PROGRAM OLD_MAIN
VAR
	fb_IndraDrive	: fbIndraDrive;
	stAmsNetId	AT %I*	: AMSNETID;
	nPort	AT %I* : WORD;
	stCommands: ST_AXIS_COMMAND;
	stStatus: ST_AXIS_STATUS;
	nMasterAxisPosition AT %I* : DINT;
	nAdditivePositionSetpoiunt AT %Q* : DINT;
	fMasterAxisPosition : LREAL;
	fAdditivePositionSetpoint : LREAL;
	fDiffPosition :LREAL;
	dLatchedPosition AT %I*:DINT;
	eTargetState: TARGET_STATE_MACHINE;
	bExecute: BOOL := FALSE;
	bEnable:BOOL:=FALSE;
	bEnabled:BOOL:=FALSE;
	bReset:BOOL:=FALSE;
    fbModePhase:FB_ModePhasing;	
	fAccelerationDefault:LREAL:=0.005;
	fSetVelToDriveRaw:LREAL;
	bBrakeFreewheelOn AT %Q*: BOOL;
	bBrakeLockedOn AT %Q*: BOOL;
    inputDummy AT %I*: BOOL;
	inputDigSens1 AT %I*: BOOL;
	inputDigSens2 AT %I*: BOOL;
	nMaxMotorTemperature: INT:= 50;
	fbBrakeTorque: FB_BrakeTorque;
	
END_VAR

stCommands.bEnableAxis :=bEnable;
stCommands.bHaltAxis :=bEnable;
bEnabled:=stStatus.bAxisEnabled;
stCommands.bCmd_ErrorReset:=bReset;

//MotorTemperatureMonitoring
IF Global_IO.iiAnalogueIn_1/10 >= nMaxMotorTemperature THEN
	bEnable:= FALSE;
	bExecute:= FALSE;
	
END_IF
			
CASE eTargetState OF 
	TARGET_STATE_MACHINE.CONSTANT_VELOCITY:
		stCommands.eMotionMode :=e_Motion_mode.eJogPositive;
		stCommands.eOperationMode:=e_Operation_mode_no.eSecondaryOpMode2;
		stCommands.fVelocityCommandValue:=0;		
	TARGET_STATE_MACHINE.POSITIONING:
		stCommands.eMotionMode :=e_Motion_mode.ePositioning;
		stCommands.eOperationMode:=e_Operation_mode_no.eSecondaryOpMode1;
	TARGET_STATE_MACHINE.PHASING:
   		fbModePhase(
			bExecute:=bExecute,
			stStatus:=	stStatus,
			dLatchedPosition:=dLatchedPosition,	
			stCommands:=stCommands);
END_CASE

IF NOT bExecute THEN
	stCommands.fVelocityCommandValue:=0;
END_IF	

IF stStatus.fActualVelocity/10 > Target_GlobalVariableList.fNominalSpeedRpm * 0.995  THEN
	stCommands.fCommandAcceleration:= fAccelerationDefault;
	stCommands.fCommandDeceleration:=fAccelerationDefault;	
ELSIF stStatus.fActualVelocity/10 > Target_GlobalVariableList.fNominalSpeedRpm * 0.9  THEN
	
	stCommands.fCommandAcceleration:= fAccelerationDefault*0.2;
	stCommands.fCommandDeceleration:=fAccelerationDefault*0.2;	
ELSIF stStatus.fActualVelocity/10 > Target_GlobalVariableList.fNominalSpeedRpm * 0.80 THEN
 	stCommands.fCommandAcceleration:= fAccelerationDefault*0.35;
	stCommands.fCommandDeceleration:=fAccelerationDefault*0.35;	
ELSIF stStatus.fActualVelocity/10 > Target_GlobalVariableList.fNominalSpeedRpm * 0.70 THEN
 	stCommands.fCommandAcceleration:= fAccelerationDefault*0.5;
	stCommands.fCommandDeceleration:=fAccelerationDefault*0.5;	
ELSE
 	stCommands.fCommandAcceleration:= fAccelerationDefault;
	stCommands.fCommandDeceleration:=fAccelerationDefault;
END_IF
IF NOT bexecute THEN
	stCommands.fCommandAcceleration:= fAccelerationDefault*4;
	stCommands.fCommandDeceleration:=fAccelerationDefault*4;
END_IF



fb_IndraDrive(
	AmsNetId:= stAmsNetId, 
	AdsAddr_Port:= nPort, 
	stAxisCommands:= stCommands, 
	stDriveStatus:= , 
	stAxisStatus=> stStatus, 
	stDriveCommands=> );
	
	stCommands.bCmd_ActivateParameterMode;//True puts the drive in parameter mode
	stCommands.bCmd_DisableLimits;// True disables monitoring of errors
	stCommands.bCmd_DriveControlledHoming;// True starts homing procedure defined in the drive
	stCommands.bCmd_ErrorReset;
	stCommands.bCmd_ExitParameterMode;
	stCommands.bCmd_RunVirtualMater;// Jog command to the virtual master
	stCommands.bCmd_SetAbsolutePosition;
	stCommands.bCommandPositionChange;// Drive moves to the current target position, when bCommandVAlueAccept toggled, drive moves to the new target position
	stCommands.bCommandValueAccept;// Used in "Drive positioning Mode" to update the target position when toggled
	stCommands.bEnableAxis;
	stCommands.bHaltAxis;// Performs halt on the drive, bEnableaxis has to be TRUE
	stCommands.bPositionCommandValue;//0=Absolute;1=Relative
	stCommands.eMotionMode;
	stCommands.eOperationMode;
	stCommands.fCommandAcceleration;// Acceleration used for positioning and jogging
	stCommands.fCommandDeceleration;// Deceleration used for positioning and jogging
	stCommands.fCommandPosition;
	stCommands.fCommandVelocity;// Velocity used for positioning and jogging
	stCommands.fFeedrateOverride;// Parameter used for adjustment of the velocity (0,100)%
	stCommands.fTorqueLimit;
	stCommands.fVelocityCommandValue;// S40, velocity used for positining and jogging (in velocity mode)
	fSetVelToDriveRaw:= DINT_TO_LREAL(MAIN.fb_IndraDrive.stDriveCommands.nS40_VelocityCommandValue)/10000;

END_PROGRAM

(* stored: Version 1.1.0.1, ProductVersion 3.1.4022.6
   POU OLD_MAIN: Id {40828a63-f1c1-40a3-a7c5-8a47be350a36}, SpecialFunc None *)
